(* 
:Description: This function block is base for all other analog devices.
*)
FUNCTION_BLOCK ABSTRACT FB_AnalogDevice IMPLEMENTS I_AnalogDevice
VAR
	sName 		: STRING; (* Name of analog device instance *)
	sModuleType : STRING; (* Name of analog device instance *)
	sPortID		: STRING; (* Slot number on the module *)
END_VAR
(*
Version history:

+-------------+------------+----------------+----------+------------------------------------------+
|Date         | Version    | created under  | Author   | Remark                                   |
+=============+============+================+==========+==========================================+
|2024-02      | 1.0.0.0    | V3.1.4024.22   | HVAP     | Function block created                   |
+-------------+------------+----------------+----------+------------------------------------------+

*)

PROPERTY ModuleType : REFERENCE TO STRING
GET
ModuleType REF= sModuleType;
END_GET
END_PROPERTY

(*
:Description: Call this method in the first cycle of the program
*)
METHOD MR_FirstCycle : BOOL
VAR_INPUT
	sName		: STRING;
	sModuleType	: STRING;
	sPortID		: STRING;
END_VAR
THIS^.sName 		:= sName;
THIS^.sModuleType 	:= sModuleType;
THIS^.sPortID 		:= sPortID;
END_METHOD

PROPERTY Name : REFERENCE TO STRING
GET
Name REF= sName;
END_GET
END_PROPERTY

PROPERTY PortID : REFERENCE TO STRING
GET
PortID REF= sPortID;
END_GET
END_PROPERTY

END_FUNCTION_BLOCK

(* stored: Version 1.1.0.1, ProductVersion 3.1.4024.9
   POU FB_AnalogDevice: Id {fd1ff737-3357-40b9-9768-3905912672c0}, SpecialFunc None
   Folder FirstCycle: Id {4838277a-937b-4d08-8eea-06187290742e}
   Folder Properties: Id {f1a577bf-52c6-4eb4-9d3c-64a214ae064d}
   Property ModuleType: Id {f871ca6f-c179-49f3-a474-2858eb824df9}
   Get Get: Id {6000fae3-4ae0-40ad-a735-38039d320380}
   Method MR_FirstCycle: Id {8f149035-58d2-427d-90ed-ab9b25d09b01}
   Property Name: Id {ff6c1a88-f757-442c-9553-e7ee63a17cd4}
   Get Get: Id {82df3994-9f25-48fa-b6e5-a43fa0761929}
   Property PortID: Id {abd8ec42-a7c1-4dec-ae55-0be5b99e9804}
   Get Get: Id {057fbfe2-5496-47fe-98e2-e12058d45dfb} *)
